Fanuc KAREL source: V_CSAPI_TESTRUN.kl

PROGRAM T
%NOLOCKGROUP
VAR
 v0 : STRING[40]
 v1 : INTEGER
 v2 : INTEGER
BEGIN
 V_CSAPI_TESTRUN(v0, v1, v2)
END T
